(* PLC project KinIn_v3.project, CODESYS CODESYS V3.5 SP19 *)
(* stored: creationDateTime 2025-01-20T16:28:46.9120419, modificationDateTime 2025-01-20T16:17:39.6822999 *)

FUNCTION_BLOCK RndStart
  VAR_INPUT
    ar_JointLimits : ARRAY[1..GVL.nJoints, 1..2] OF REAL;
  END_VAR
  VAR_OUTPUT
    randomArray : ARRAY[1..GVL.nJoints] OF REAL;
  END_VAR
  VAR
    i : DINT;  (* RndFunc:RDM;//OSCAT_BASIC.RDM; *)
    rndNum : REAL;
    rndNum_scaled : REAL;
    maxVal : REAL;
    minVal : REAL;
    scale : REAL;
    meanVal : REAL;
  END_VAR

            //robot limits in  degrees
//give lenghts and create the Vb for forward and bacward 
rndNum:=0;
FOR i:=1 TO GVL.nJoints DO
	maxVal:=ar_JointLimits[i,2];
	minVal:=ar_JointLimits[i,1];
	scale:=maxVal-minVal;
	meanVal:=(ar_JointLimits[i,2]+ar_JointLimits[i,1])/2;
	
	rndNum:=OSCAT_BASIC.RDM(last:=rndNum );
	rndNum_scaled:=rndNum*scale+meanVal;
	
	randomArray[i]:=rndNum_scaled;
END_FOR





          
END_FUNCTION_BLOCK
